(* IEC 61131-3 sources: PortalRobot/Portal_robot/Device/application (part 5) *)

(* ---- PLC_PRG.RunTestControl.st ---- *)
METHOD PRIVATE RunTestControl

// --- BEGIN IMPLEMENTATION ---

// Test environment is independent from the robot control interface.
rtTestEnvironmentApply(CLK := GVL_HMI.xTestEnvironmentApply);
rtTestSpeedProfileApply(CLK := GVL_HMI.xTestSpeedProfileApply);
rtTestScenarioApply(CLK := GVL_HMI.xTestScenarioApply);
xTestInitializePulse := FALSE;
xTestAbortActive := GVL_HMI.xTestAbort
	AND GVL_HMI.xTestSessionActive
	AND (GVL_CELL_SETTINGS.eTestEnvironment = E_CELL_TEST_ENVIRONMENT.SIMULATION);

xTestStable := NOT GVL_CELL_MANAGER.Status.xRunning
	AND NOT GVL_ROBOT.Status.xBusy
	AND NOT GVL_MAGAZINE.astStatus[1].xBusy
	AND NOT GVL_MAGAZINE.astStatus[2].xBusy
	AND NOT GVL_TWO_PALLET.astInput[1].xPowered
	AND NOT GVL_TWO_PALLET.astInput[2].xPowered
	AND NOT xMotionBusy
	AND NOT SIMULATION_DYNAMICS.xBusy;
FOR uiTestIndex := UINT#1 TO UINT#3 DO
	xTestStable := xTestStable
		AND NOT GVL_MACHINE.Status[uiTestIndex].xBusy
		AND NOT GVL_MACHINE.Status[uiTestIndex].xProcessing;
END_FOR;

GVL_HMI.xTestEnvironmentChangeAllowed := xTestStable;
GVL_HMI.xTestScenarioApplyAllowed := xTestStable
	AND (GVL_TWO_PALLET.uiMode = 0) // Existing scenarios describe static 120-slot magazines
	AND GVL_HMI.xTestSessionActive
	AND (GVL_CELL_SETTINGS.eTestEnvironment <> E_CELL_TEST_ENVIRONMENT.NORMAL)
	AND ((GVL_CELL_SETTINGS.eTestEnvironment <> E_CELL_TEST_ENVIRONMENT.SC500_BENCH)
		OR GVL_TEST_IO.xSc500BenchKeyInput)
	AND ((GVL_CELL_SETTINGS.eTestEnvironment <> E_CELL_TEST_ENVIRONMENT.SIMULATION)
		OR NOT GVL_ROBOT_MODBUS.xModeActive
		OR GVL_ROBOT_MODBUS.Status.xSimulatorActive);
GVL_HMI.xSc500BenchKeyActive := GVL_TEST_IO.xSc500BenchKeyInput;

IF rtTestEnvironmentApply.Q THEN
	GVL_HMI.uiTestRejectReason := UINT#0;
	IF NOT GVL_HMI.xTestEnvironmentChangeAllowed THEN
		GVL_HMI.uiTestRejectReason := UINT#1; // equipment is not idle
	ELSIF GVL_HMI.uiTestEnvironmentRequest > UINT#2 THEN
		GVL_HMI.uiTestRejectReason := UINT#2; // invalid environment
	ELSIF (GVL_HMI.uiTestEnvironmentRequest = UINT#2)
	AND (NOT GVL_ROBOT_MODBUS.xModeActive OR NOT GVL_TEST_IO.xSc500BenchKeyInput) THEN
		GVL_HMI.uiTestRejectReason := UINT#3; // bench requires Modbus and physical key
	ELSIF (GVL_HMI.uiTestEnvironmentRequest = UINT#1)
	AND GVL_ROBOT_MODBUS.xModeActive
	AND NOT GVL_ROBOT_MODBUS.Status.xSimulatorActive THEN
		GVL_HMI.uiTestRejectReason := UINT#4; // Python simulator marker missing
	ELSE
		CASE GVL_HMI.uiTestEnvironmentRequest OF
			UINT#0: GVL_CELL_SETTINGS.eTestEnvironment := E_CELL_TEST_ENVIRONMENT.NORMAL;
			UINT#1: GVL_CELL_SETTINGS.eTestEnvironment := E_CELL_TEST_ENVIRONMENT.SIMULATION;
			UINT#2: GVL_CELL_SETTINGS.eTestEnvironment := E_CELL_TEST_ENVIRONMENT.SC500_BENCH;
		END_CASE;
		GVL_CELL_SETTINGS.eTestSpeedProfile := E_TEST_SPEED_PROFILE.REALTIME;
		xSc500BenchKeyLost := FALSE;
	END_IF;
END_IF;

IF rtTestSpeedProfileApply.Q THEN
	GVL_HMI.uiTestRejectReason := UINT#0;
	IF (GVL_HMI.uiTestSpeedProfileRequest <= UINT#1)
	AND (GVL_CELL_SETTINGS.eTestEnvironment = E_CELL_TEST_ENVIRONMENT.SIMULATION) THEN
		IF GVL_HMI.uiTestSpeedProfileRequest = UINT#1 THEN
			GVL_CELL_SETTINGS.eTestSpeedProfile := E_TEST_SPEED_PROFILE.FAST;
			// В Modbus профиль по-прежнему владеет коэффициентом внешней модели.
			// В SoftMotion коэффициент задаёт ползунок, а применение выполняется
			// отдельной транзакцией только на границе следующего теста.
			IF GVL_ROBOT_MODBUS.xModeActive THEN
				GVL_CELL_SETTINGS.uiSimulationTimeFactor := UINT#250;
			END_IF;
		ELSE
			GVL_CELL_SETTINGS.eTestSpeedProfile := E_TEST_SPEED_PROFILE.REALTIME;
			IF GVL_ROBOT_MODBUS.xModeActive THEN
				GVL_CELL_SETTINGS.uiSimulationTimeFactor := UINT#1;
			END_IF;
		END_IF;
		GVL_HMI.uiSimulationTimeFactor := GVL_CELL_SETTINGS.uiSimulationTimeFactor;
	ELSE
		GVL_HMI.uiTestRejectReason := UINT#5; // speed profile is simulation-only
	END_IF;
END_IF;

// Losing the physical key does not interrupt the current SC-500 command.
// As soon as it finishes, robot readiness is removed and no next command can start.
IF (GVL_CELL_SETTINGS.eTestEnvironment = E_CELL_TEST_ENVIRONMENT.SC500_BENCH)
AND NOT GVL_TEST_IO.xSc500BenchKeyInput THEN
	xSc500BenchKeyLost := TRUE;
	IF NOT GVL_ROBOT_MODBUS.Status.xBusy THEN
		xRobotInterfaceReady := FALSE;
		xDrivesReady := FALSE;
	END_IF;
END_IF;

IF rtTestScenarioApply.Q THEN
	GVL_HMI.uiTestScenarioResult := UINT#0;
	xTestScenarioValid := GVL_HMI.stTestScenario.udiLoadSeq <> UDINT#0
		AND (GVL_HMI.stTestScenario.uiTypeCount >= UINT#1)
		AND (GVL_HMI.stTestScenario.uiTypeCount <= UINT#3);
	FOR uiTestIndex := UINT#1 TO UINT#3 DO
		xTestScenarioValid := xTestScenarioValid
			AND (GVL_HMI.stTestScenario.auiMachineState[uiTestIndex] <= UINT#3)
			AND (GVL_HMI.stTestScenario.auiMachineType[uiTestIndex] >= UINT#1)
			AND (GVL_HMI.stTestScenario.auiMachineType[uiTestIndex]
				<= GVL_HMI.stTestScenario.uiTypeCount);
	END_FOR;
	FOR uiTestIndex := UINT#1 TO UINT#120 DO
		xTestScenarioValid := xTestScenarioValid
			AND (GVL_HMI.stTestScenario.auiSlotType[uiTestIndex] >= UINT#1)
			AND (GVL_HMI.stTestScenario.auiSlotType[uiTestIndex]
				<= GVL_HMI.stTestScenario.uiTypeCount);
		FOR uiTestMagazine := UINT#1 TO UINT#2 DO
			xTestScenarioValid := xTestScenarioValid
				AND (GVL_HMI.stTestScenario.aauiSlotContent[uiTestMagazine, uiTestIndex] <= UINT#2);
		END_FOR;
	END_FOR;
	uiTestFaultOwnerCount := UINT#0;
	IF GVL_HMI.stTestScenario.dwCellFaultMask <> DWORD#0 THEN
		uiTestFaultOwnerCount := uiTestFaultOwnerCount + UINT#1;
	END_IF;
	IF GVL_HMI.stTestScenario.dwRobotFaultMask <> DWORD#0 THEN
		uiTestFaultOwnerCount := uiTestFaultOwnerCount + UINT#1;
	END_IF;
	FOR uiTestMagazine := UINT#1 TO UINT#2 DO
		IF GVL_HMI.stTestScenario.adwMagazineFaultMask[uiTestMagazine] <> DWORD#0 THEN
			uiTestFaultOwnerCount := uiTestFaultOwnerCount + UINT#1;
		END_IF;
		xTestScenarioValid := xTestScenarioValid
			AND (GVL_HMI.stTestScenario.adwMagazineFaultMask[uiTestMagazine] <= DWORD#16#0000_003F);
	END_FOR;
	FOR uiTestIndex := UINT#1 TO UINT#3 DO
		IF GVL_HMI.stTestScenario.adwMachineFaultMask[uiTestIndex] <> DWORD#0 THEN
			uiTestFaultOwnerCount := uiTestFaultOwnerCount + UINT#1;
		END_IF;
		xTestScenarioValid := xTestScenarioValid
			AND (GVL_HMI.stTestScenario.adwMachineFaultMask[uiTestIndex] <= DWORD#16#0000_07FF);
	END_FOR;
	xTestScenarioValid := xTestScenarioValid
		AND (uiTestFaultOwnerCount <= UINT#1)
		AND (GVL_HMI.stTestScenario.dwCellFaultMask <= DWORD#16#0000_0001)
		AND (GVL_HMI.stTestScenario.dwRobotFaultMask <= DWORD#16#0000_01FF)
		AND (GVL_HMI.stTestScenario.auiGripperContent[1] <= UINT#1)
		AND ((GVL_HMI.stTestScenario.auiGripperContent[1] = UINT#0)
			= (GVL_HMI.stTestScenario.auiGripperType[1] = UINT#0))
		AND (GVL_HMI.stTestScenario.auiGripperType[1]
			<= GVL_HMI.stTestScenario.uiTypeCount)
		AND ((GVL_HMI.stTestScenario.auiGripperContent[2] = UINT#0)
			OR (GVL_HMI.stTestScenario.auiGripperContent[2] = UINT#2))
		AND ((GVL_HMI.stTestScenario.auiGripperContent[2] = UINT#0)
			= (GVL_HMI.stTestScenario.auiGripperType[2] = UINT#0))
		AND (GVL_HMI.stTestScenario.auiGripperType[2]
			<= GVL_HMI.stTestScenario.uiTypeCount);

	IF NOT GVL_HMI.xTestScenarioApplyAllowed THEN
		GVL_HMI.uiTestScenarioResult := UINT#1;
	ELSIF NOT xTestScenarioValid OR (GVL_HMI.stTestScenario.uiOrientation > UINT#1) THEN
		GVL_HMI.uiTestScenarioResult := UINT#2;
	ELSE
		FOR uiTestMagazine := UINT#1 TO UINT#2 DO
			FOR uiTestIndex := UINT#1 TO UINT#120 DO
				GVL_DETAIL.astMagazine[uiTestMagazine].aSlots[uiTestIndex].xInPosition :=
					GVL_HMI.stTestScenario.aauiSlotContent[uiTestMagazine, uiTestIndex] <> UINT#0;
				CASE GVL_HMI.stTestScenario.aauiSlotContent[uiTestMagazine, uiTestIndex] OF
					UINT#1: GVL_DETAIL.astMagazine[uiTestMagazine].aSlots[uiTestIndex].eDetailType := E_DETAIL_TYPE.BLANK;
					UINT#2: GVL_DETAIL.astMagazine[uiTestMagazine].aSlots[uiTestIndex].eDetailType := E_DETAIL_TYPE.DETAIL;
				ELSE
					GVL_DETAIL.astMagazine[uiTestMagazine].aSlots[uiTestIndex].eDetailType := E_DETAIL_TYPE.NONE;
				END_CASE;
				IF GVL_HMI.stTestScenario.aauiSlotContent[uiTestMagazine, uiTestIndex] = UINT#0 THEN
					GVL_DETAIL.astMagazine[uiTestMagazine].aSlots[uiTestIndex].uiProductType := UINT#0;
				ELSE
					GVL_DETAIL.astMagazine[uiTestMagazine].aSlots[uiTestIndex].uiProductType :=
						GVL_HMI.stTestScenario.auiSlotType[uiTestIndex];
				END_IF;
			END_FOR;
			adwTestMagazineFaultMask[uiTestMagazine] :=
				GVL_HMI.stTestScenario.adwMagazineFaultMask[uiTestMagazine];
		END_FOR;
		// Начальные инъекции: маски переводятся в существующий диагностический
		// контракт, а не обходят владельцев ошибок.
		axHmiInternalPulse[13] :=
			(GVL_HMI.stTestScenario.dwCellFaultMask AND DWORD#16#0000_0001) <> DWORD#0;
		axHmiInternalPulse[12] :=
			(GVL_HMI.stTestScenario.dwRobotFaultMask AND DWORD#16#0000_0001) <> DWORD#0;
		GVL_HMI.xSimGripper1Fault :=
			(GVL_HMI.stTestScenario.dwRobotFaultMask AND DWORD#16#0000_0002) <> DWORD#0;
		GVL_HMI.xSimGripper2Fault :=
			(GVL_HMI.stTestScenario.dwRobotFaultMask AND DWORD#16#0000_0004) <> DWORD#0;
		GVL_HMI.xSimGripperRotationFault :=
			(GVL_HMI.stTestScenario.dwRobotFaultMask AND DWORD#16#0000_0008) <> DWORD#0;
		GVL_HMI.xSimGripperGlobalFault :=
			(GVL_HMI.stTestScenario.dwRobotFaultMask AND DWORD#16#0000_0010) <> DWORD#0;
		axHmiInternalPulse[14] :=
			(GVL_HMI.stTestScenario.dwRobotFaultMask AND DWORD#16#0000_0020) <> DWORD#0;
		axHmiInternalPulse[15] :=
			(GVL_HMI.stTestScenario.dwRobotFaultMask AND DWORD#16#0000_0040) <> DWORD#0;
		axHmiInternalPulse[16] :=
			(GVL_HMI.stTestScenario.dwRobotFaultMask AND DWORD#16#0000_0080) <> DWORD#0;
		axHmiInternalPulse[17] :=
			(GVL_HMI.stTestScenario.dwRobotFaultMask AND DWORD#16#0000_0100) <> DWORD#0;
		axHmiInternalPulse[18] :=
			(GVL_HMI.stTestScenario.adwMagazineFaultMask[1] AND DWORD#16#0000_0001) <> DWORD#0;
		axHmiInternalPulse[19] :=
			(GVL_HMI.stTestScenario.adwMagazineFaultMask[1] AND DWORD#16#0000_0002) <> DWORD#0;
		axHmiInternalPulse[20] :=
			(GVL_HMI.stTestScenario.adwMagazineFaultMask[1] AND DWORD#16#0000_0004) <> DWORD#0;
		axHmiInternalPulse[21] :=
			(GVL_HMI.stTestScenario.adwMagazineFaultMask[1] AND DWORD#16#0000_0008) <> DWORD#0;
		axHmiInternalPulse[22] :=
			(GVL_HMI.stTestScenario.adwMagazineFaultMask[1] AND DWORD#16#0000_0010) <> DWORD#0;
		axHmiInternalPulse[23] :=
			(GVL_HMI.stTestScenario.adwMagazineFaultMask[1] AND DWORD#16#0000_0020) <> DWORD#0;
		FOR uiTestIndex := UINT#1 TO UINT#3 DO
			GVL_HMI.axMachineSimAlarm[uiTestIndex] :=
				(GVL_HMI.stTestScenario.adwMachineFaultMask[uiTestIndex] AND DWORD#16#0000_0001) <> DWORD#0;
			GVL_HMI.axMachineSimDoorFault[uiTestIndex] :=
				(GVL_HMI.stTestScenario.adwMachineFaultMask[uiTestIndex] AND DWORD#16#0000_0002) <> DWORD#0;
			GVL_HMI.axMachineSimChuckFault[uiTestIndex] :=
				(GVL_HMI.stTestScenario.adwMachineFaultMask[uiTestIndex] AND DWORD#16#0000_0004) <> DWORD#0;
			GVL_HMI.axMachineTimeoutRobotMove[uiTestIndex] :=
				(GVL_HMI.stTestScenario.adwMachineFaultMask[uiTestIndex] AND DWORD#16#0000_0008) <> DWORD#0;
			GVL_HMI.axMachineTimeoutRobotAction[uiTestIndex] :=
				(GVL_HMI.stTestScenario.adwMachineFaultMask[uiTestIndex] AND DWORD#16#0000_0010) <> DWORD#0;
			GVL_HMI.axMachineTimeoutRobotRelease[uiTestIndex] :=
				(GVL_HMI.stTestScenario.adwMachineFaultMask[uiTestIndex] AND DWORD#16#0000_0020) <> DWORD#0;
			GVL_HMI.axMachineTimeoutDoorOpen[uiTestIndex] :=
				(GVL_HMI.stTestScenario.adwMachineFaultMask[uiTestIndex] AND DWORD#16#0000_0040) <> DWORD#0;
			GVL_HMI.axMachineTimeoutDoorClose[uiTestIndex] :=
				(GVL_HMI.stTestScenario.adwMachineFaultMask[uiTestIndex] AND DWORD#16#0000_0080) <> DWORD#0;
			GVL_HMI.axMachineTimeoutChuckOpen[uiTestIndex] :=
				(GVL_HMI.stTestScenario.adwMachineFaultMask[uiTestIndex] AND DWORD#16#0000_0100) <> DWORD#0;
			GVL_HMI.axMachineTimeoutChuckClose[uiTestIndex] :=
				(GVL_HMI.stTestScenario.adwMachineFaultMask[uiTestIndex] AND DWORD#16#0000_0200) <> DWORD#0;
			GVL_HMI.axMachineTimeoutCycleStart[uiTestIndex] :=
				(GVL_HMI.stTestScenario.adwMachineFaultMask[uiTestIndex] AND DWORD#16#0000_0400) <> DWORD#0;
		END_FOR;
		GVL_HMI.xErrorSimulationEnable :=
			(GVL_HMI.stTestScenario.dwCellFaultMask <> DWORD#0)
			OR (GVL_HMI.stTestScenario.dwRobotFaultMask <> DWORD#0)
			OR (GVL_HMI.stTestScenario.adwMagazineFaultMask[1] <> DWORD#0)
			OR (GVL_HMI.stTestScenario.adwMagazineFaultMask[2] <> DWORD#0)
			OR (GVL_HMI.stTestScenario.adwMachineFaultMask[1] <> DWORD#0)
			OR (GVL_HMI.stTestScenario.adwMachineFaultMask[2] <> DWORD#0)
			OR (GVL_HMI.stTestScenario.adwMachineFaultMask[3] <> DWORD#0);
		xTestInitializePulse := TRUE;
	END_IF;
	// Ack подтверждает обработку конкретного LoadSeq даже при отклонении.
	GVL_HMI.udiTestScenarioAckSeq := GVL_HMI.stTestScenario.udiLoadSeq;
END_IF;

GVL_HMI.uiTestEnvironmentApplied := TO_UINT(GVL_CELL_SETTINGS.eTestEnvironment);
GVL_HMI.uiTestSpeedProfileApplied := TO_UINT(GVL_CELL_SETTINGS.eTestSpeedProfile);
GVL_HMI.xSc500BenchKeyLost := xSc500BenchKeyLost;
IF GVL_CELL_SETTINGS.eTestEnvironment = E_CELL_TEST_ENVIRONMENT.SIMULATION THEN
	IF GVL_HMI.xTestSessionActive THEN
		GVL_CELL_SETTINGS.xSimulationAccelerationEnable :=
			GVL_CELL_SETTINGS.eTestSpeedProfile = E_TEST_SPEED_PROFILE.FAST;
		// Профиль владеет включением ускоренных таймеров, а сам коэффициент
		// разрешено менять с HMI прямо во время тестового движения.
		GVL_HMI.xSimulationAccelerationEnable := GVL_CELL_SETTINGS.xSimulationAccelerationEnable;
	END_IF;
ELSE
	GVL_CELL_SETTINGS.xSimulationAccelerationEnable := FALSE;
	GVL_HMI.xSimulationAccelerationEnable := FALSE;
END_IF;

(* ---- PLC_PRG.RunTwoPallet.st ---- *)
METHOD PRIVATE RunTwoPallet

// --- BEGIN IMPLEMENTATION ---

GVL_TWO_PALLET.xModeChanged := FALSE;
IF NOT xTwinSimulationInitialized THEN
	FOR uiTwin := 1 TO 2 DO
		// Числа используются только для виртуальных SoftMotion-осей.
		GVL_TWO_PALLET.astSimulationConfig[uiTwin].xConfigured := TRUE;
		GVL_TWO_PALLET.astSimulationConfig[uiTwin].xP1LockOut := TRUE;
		GVL_TWO_PALLET.axSimulationAutoSwapEnabled[uiTwin] := TRUE;
		GVL_TWO_PALLET.astSimulationConfig[uiTwin].lrExchange := 0.0;
		GVL_TWO_PALLET.astSimulationConfig[uiTwin].lrWorkP1 := 100.0;
		GVL_TWO_PALLET.astSimulationConfig[uiTwin].lrWorkP2 := 200.0;
		GVL_TWO_PALLET.astSimulationConfig[uiTwin].lrHome := 0.0;
		GVL_TWO_PALLET.astSimulationConfig[uiTwin].lrTolerance := 1.0;
		GVL_TWO_PALLET.astSimulationConfig[uiTwin].lrVelocity := 100.0;
		GVL_TWO_PALLET.astSimulationConfig[uiTwin].lrAcceleration := 200.0;
		GVL_TWO_PALLET.astSimulationConfig[uiTwin].lrDeceleration := 200.0;
		GVL_TWO_PALLET.astSimulationConfig[uiTwin].lrJerk := 1000.0;
		GVL_TWO_PALLET.astSimulationConfig[uiTwin].tCylinder := T#3S;
		GVL_TWO_PALLET.astSimulationConfig[uiTwin].tMove := T#20S;
		GVL_TWO_PALLET.astSimulationConfig[uiTwin].tHome := T#10S;
		GVL_TWO_PALLET.astSimulationConfig[uiTwin].tPulse := T#150MS;
	END_FOR;
	IF NOT GVL_TWO_PALLET.xAutoSwapDefaultsApplied THEN
		FOR uiTwin := 1 TO 2 DO
			GVL_TWO_PALLET.axAutoSwapEnabled[uiTwin] := TRUE;
		END_FOR;
		GVL_TWO_PALLET.xAutoSwapDefaultsApplied := TRUE;
	END_IF;
	xTwinSimulationInitialized := TRUE;
END_IF;
FOR uiTwin := 1 TO 2 DO
	GVL_TWO_PALLET.auiCommand[uiTwin] := UINT#0;
END_FOR;
IF NOT xTwinStartup THEN
	IF GVL_TWO_PALLET.uiMode = 0 THEN
		GVL_HMI.MagazinePitchX := GVL_TWO_PALLET.lrStaticPitchX;
		GVL_HMI.MagazinePitchY := GVL_TWO_PALLET.lrStaticPitchY;
	ELSE
		GVL_HMI.MagazinePitchX := GVL_TWO_PALLET.lrTwinPitchX;
		GVL_HMI.MagazinePitchY := GVL_TWO_PALLET.lrTwinPitchY;
	END_IF;
	FOR uiTwin := 1 TO 2 DO
		// После перезапуска содержимое сохранено, готовность загрузки подтверждается заново.
		GVL_TWO_PALLET.astStore[uiTwin].axLoaded[1] := FALSE;
		GVL_TWO_PALLET.astStore[uiTwin].axLoaded[2] := FALSE;
		IF GVL_TWO_PALLET.uiMode = 0 THEN
			GVL_DETAIL.astMagazine[uiTwin] := GVL_TWO_PALLET.astStatic[uiTwin];
		END_IF;
	END_FOR;
	xTwinStartup := TRUE;
END_IF;
GVL_TWO_PALLET.xModeChangeAllowed := GVL_CELL_CONTROL.xManual
	AND NOT GVL_CELL_MANAGER.Status.xRunning AND NOT GVL_ROBOT.Status.xBusy AND NOT xMotionBusy
	AND xHmiConnectionAlive AND NOT GVL_HMI.xTestSessionActive AND NOT GVL_ROBOT.Status.xBlankAvailable AND NOT GVL_ROBOT.Status.xDetailAvailable
	AND (GVL_ROBOT.Status.uiMagazineContext = 0)
	AND NOT GVL_MAGAZINE.astStatus[1].xEnabled AND NOT GVL_MAGAZINE.astStatus[2].xEnabled
	AND NOT GVL_MAGAZINE.astStatus[1].xBusy AND NOT GVL_MAGAZINE.astStatus[2].xBusy
	AND NOT GVL_TWO_PALLET.astStatus[1].xBusy AND NOT GVL_TWO_PALLET.astStatus[2].xBusy
	AND NOT GVL_TWO_PALLET.astInput[1].xPowered AND NOT GVL_TWO_PALLET.astInput[2].xPowered
	AND NOT GVL_TWO_PALLET.astStatus[1].xError AND NOT GVL_TWO_PALLET.astStatus[2].xError;

udiTwinSnapshot := GVL_HMI.udiTwinCommandSeq;
uiTwinRequestResult := 0;
xTwinInventoryCommand := FALSE;
IF (udiTwinSnapshot <> 0) AND (udiTwinSnapshot <> GVL_HMI.udiTwinAckSeq) THEN
	stTwinRequest := GVL_HMI.stTwinRequest;
	uiTwinRequestResult := 2; // Условие команды не выполнено
	IF (GVL_HMI.udiHmiCommandClockMs - GVL_HMI.udiTwinIssuedAtMs) > 2000 THEN
		uiTwinRequestResult := 4;
	ELSIF (stTwinRequest.uiMagazine = 0) AND (stTwinRequest.uiCommand = 25) THEN
		IF GVL_TWO_PALLET.xModeChangeAllowed AND (stTwinRequest.uiValue <= 1) AND xHmiConnectionAlive THEN
			IF GVL_TWO_PALLET.uiMode <> stTwinRequest.uiValue THEN
				IF GVL_TWO_PALLET.uiMode = 0 THEN
					GVL_TWO_PALLET.lrStaticPitchX := GVL_HMI.MagazinePitchX;
					GVL_TWO_PALLET.lrStaticPitchY := GVL_HMI.MagazinePitchY;
				ELSE
					GVL_TWO_PALLET.lrTwinPitchX := GVL_HMI.MagazinePitchX;
					GVL_TWO_PALLET.lrTwinPitchY := GVL_HMI.MagazinePitchY;
				END_IF;
				GVL_TWO_PALLET.uiMode := stTwinRequest.uiValue;
				GVL_TWO_PALLET.xModeChanged := TRUE;
				FOR uiTwin := 1 TO 2 DO
					IF GVL_TWO_PALLET.uiMode = 0 THEN GVL_DETAIL.astMagazine[uiTwin] := GVL_TWO_PALLET.astStatic[uiTwin]; END_IF;
					// Базы меняются вместе с механикой: старые координаты нельзя молча использовать.
					GVL_POINT.astRetainPoints[13 + uiTwin].xConfigured := FALSE;
				END_FOR;
				IF GVL_TWO_PALLET.uiMode = 0 THEN
					GVL_HMI.MagazinePitchX := GVL_TWO_PALLET.lrStaticPitchX; GVL_HMI.MagazinePitchY := GVL_TWO_PALLET.lrStaticPitchY;
				ELSE
					GVL_HMI.MagazinePitchX := GVL_TWO_PALLET.lrTwinPitchX; GVL_HMI.MagazinePitchY := GVL_TWO_PALLET.lrTwinPitchY;
				END_IF;
				xPointTableReady := FALSE;
			END_IF;
			uiTwinRequestResult := 1;
		END_IF;
	ELSIF (stTwinRequest.uiMagazine >= 1) AND (stTwinRequest.uiMagazine <= 2)
		AND (GVL_TWO_PALLET.uiMode = 1) THEN
		uiTwin := stTwinRequest.uiMagazine;
		IF ((stTwinRequest.uiCommand >= 1) AND (stTwinRequest.uiCommand <= 19))
			OR ((stTwinRequest.uiCommand >= 25) AND (stTwinRequest.uiCommand <= 32)) THEN
			GVL_TWO_PALLET.auiCommand[uiTwin] := stTwinRequest.uiCommand;
			GVL_TWO_PALLET.auiValue[uiTwin] := stTwinRequest.uiValue;
			GVL_TWO_PALLET.audiRevision[uiTwin] := stTwinRequest.udiRevision;
		ELSIF (stTwinRequest.uiCommand >= UINT#20)
			AND (stTwinRequest.uiCommand <= UINT#24) THEN
			xTwinInventoryCommand := TRUE; // Проверить по разрешениям текущего скана ПОСЛЕ вызова FB
		ELSIF stTwinRequest.uiCommand = UINT#33 THEN
			IF (stTwinRequest.uiValue <= UINT#1) AND xHmiConnectionAlive THEN
				IF GVL_CELL_SETTINGS.eTestEnvironment = E_CELL_TEST_ENVIRONMENT.SIMULATION THEN
					GVL_TWO_PALLET.axSimulationAutoSwapEnabled[uiTwin] := stTwinRequest.uiValue = UINT#1;
				ELSE
					GVL_TWO_PALLET.axAutoSwapEnabled[uiTwin] := stTwinRequest.uiValue = UINT#1;
				END_IF;
				uiTwinRequestResult := UINT#1;
			END_IF;
		END_IF;
	END_IF;
END_IF;

FOR uiTwin := 1 TO 2 DO
	GVL_TWO_PALLET.astActiveConfig[uiTwin] := GVL_TWO_PALLET.astConfig[uiTwin];
	IF GVL_CELL_SETTINGS.eTestEnvironment = E_CELL_TEST_ENVIRONMENT.SIMULATION THEN
		GVL_TWO_PALLET.astActiveConfig[uiTwin] := GVL_TWO_PALLET.astSimulationConfig[uiTwin];
		xTwinAutoSwapEnabled := GVL_TWO_PALLET.axSimulationAutoSwapEnabled[uiTwin];
	ELSE
		xTwinAutoSwapEnabled := GVL_TWO_PALLET.axAutoSwapEnabled[uiTwin];
	END_IF;
	// Старые RETAIN-параметры сохраняют прежнюю полярность до первой настройки
	// полных сочетаний. Нормализуем только рабочую копию, без записи в RETAIN.
	IF NOT GVL_TWO_PALLET.astActiveConfig[uiTwin].xSignalPatternsConfigured THEN
		GVL_TWO_PALLET.astActiveConfig[uiTwin].uiP1Signals := UINT#38;
		GVL_TWO_PALLET.astActiveConfig[uiTwin].uiP2Signals := UINT#26;
		IF GVL_TWO_PALLET.astActiveConfig[uiTwin].xP1LockOut THEN
			GVL_TWO_PALLET.astActiveConfig[uiTwin].uiP1Signals := UINT#26;
			GVL_TWO_PALLET.astActiveConfig[uiTwin].uiP2Signals := UINT#38;
		END_IF;
		GVL_TWO_PALLET.astActiveConfig[uiTwin].xSignalPatternsConfigured := TRUE;
	END_IF;
	// Legacy power/reset также проходит владельца механизма и его блокировки.
	IF (GVL_TWO_PALLET.auiCommand[uiTwin] = 0) AND (GVL_TWO_PALLET.uiMode = 1) THEN
		IF GVL_HMI.astMagazineCommand[uiTwin].xEnable THEN GVL_TWO_PALLET.auiCommand[uiTwin] := 1; END_IF;
		IF GVL_HMI.astMagazineCommand[uiTwin].xDisable OR GVL_CELL_CONTROL.xDisable THEN GVL_TWO_PALLET.auiCommand[uiTwin] := 3; END_IF;
		IF GVL_HMI.astMagazineCommand[uiTwin].xStop THEN GVL_TWO_PALLET.auiCommand[uiTwin] := 15; END_IF;
		IF GVL_HMI.astMagazineCommand[uiTwin].xReset
			OR (GVL_CELL_CONTROL.xReset AND GVL_TWO_PALLET.astStatus[uiTwin].xResetAllowed) THEN
			GVL_TWO_PALLET.auiCommand[uiTwin] := 16;
		END_IF;
	END_IF;

	// Единственное место преобразования транспортных номеров HMI в интерфейс FB.
	astTwinCommand[uiTwin].xEnable := GVL_TWO_PALLET.auiCommand[uiTwin] = UINT#1;
	astTwinCommand[uiTwin].xConfirm := GVL_TWO_PALLET.auiCommand[uiTwin] = UINT#2;
	astTwinCommand[uiTwin].xStart := GVL_TWO_PALLET.auiCommand[uiTwin] = UINT#27;
	astTwinCommand[uiTwin].xRejectStart := GVL_TWO_PALLET.auiCommand[uiTwin] = UINT#28;
	astTwinCommand[uiTwin].xDisable := GVL_TWO_PALLET.auiCommand[uiTwin] = UINT#3;
	astTwinCommand[uiTwin].xSwap := GVL_TWO_PALLET.auiCommand[uiTwin] = UINT#4;
	astTwinCommand[uiTwin].xPowerOn := GVL_TWO_PALLET.auiCommand[uiTwin] = UINT#5;
	astTwinCommand[uiTwin].xPowerOff := GVL_TWO_PALLET.auiCommand[uiTwin] = UINT#6;
	astTwinCommand[uiTwin].xDriveReset := GVL_TWO_PALLET.auiCommand[uiTwin] = UINT#7;
	astTwinCommand[uiTwin].xHome := GVL_TWO_PALLET.auiCommand[uiTwin] = UINT#8;
	astTwinCommand[uiTwin].xLower := GVL_TWO_PALLET.auiCommand[uiTwin] = UINT#9;
	astTwinCommand[uiTwin].xRaise := GVL_TWO_PALLET.auiCommand[uiTwin] = UINT#10;
	astTwinCommand[uiTwin].xSelectPallet := (GVL_TWO_PALLET.auiCommand[uiTwin] = UINT#11)
		OR (GVL_TWO_PALLET.auiCommand[uiTwin] = UINT#12);
	astTwinCommand[uiTwin].xLockIn := GVL_TWO_PALLET.auiCommand[uiTwin] = UINT#29;
	astTwinCommand[uiTwin].xLockOut := GVL_TWO_PALLET.auiCommand[uiTwin] = UINT#30;
	astTwinCommand[uiTwin].xStopIn := GVL_TWO_PALLET.auiCommand[uiTwin] = UINT#31;
	astTwinCommand[uiTwin].xStopOut := GVL_TWO_PALLET.auiCommand[uiTwin] = UINT#32;
	astTwinCommand[uiTwin].xMoveToExchange := GVL_TWO_PALLET.auiCommand[uiTwin] = UINT#13;
	astTwinCommand[uiTwin].xMoveToWork := GVL_TWO_PALLET.auiCommand[uiTwin] = UINT#14;
	astTwinCommand[uiTwin].xStop := GVL_TWO_PALLET.auiCommand[uiTwin] = UINT#15;
	astTwinCommand[uiTwin].xReset := GVL_TWO_PALLET.auiCommand[uiTwin] = UINT#16;
	astTwinCommand[uiTwin].xJogPositive := GVL_TWO_PALLET.auiCommand[uiTwin] = UINT#17;
	astTwinCommand[uiTwin].xJogNegative := GVL_TWO_PALLET.auiCommand[uiTwin] = UINT#18;
	astTwinCommand[uiTwin].xJogRelease := GVL_TWO_PALLET.auiCommand[uiTwin] = UINT#19;
	astTwinCommand[uiTwin].xTeachOperator := GVL_TWO_PALLET.auiCommand[uiTwin] = UINT#25;
	astTwinCommand[uiTwin].xTeachWork := GVL_TWO_PALLET.auiCommand[uiTwin] = UINT#26;
	astTwinCommand[uiTwin].uiPallet := GVL_TWO_PALLET.auiValue[uiTwin];
	IF GVL_TWO_PALLET.auiCommand[uiTwin] = UINT#11 THEN
		astTwinCommand[uiTwin].uiPallet := UINT#1;
	ELSIF GVL_TWO_PALLET.auiCommand[uiTwin] = UINT#12 THEN
		astTwinCommand[uiTwin].uiPallet := UINT#2;
	END_IF;
	astTwinCommand[uiTwin].udiRevision := GVL_TWO_PALLET.audiRevision[uiTwin];

	// xBusy не покрывает удерживаемый запрос и завершение Disable.
	// Занятость другого магазина/станка сама по себе не запрещает правку инвентаря.
	xTwinRobotOperation := GVL_MAGAZINE.astPartStatus[uiTwin].xBusy
		OR GVL_MAGAZINE.astPartStatus[uiTwin].xDisablePending
		OR GVL_MAGAZINE.astAutoCommand[uiTwin].xExecute
		OR GVL_MAGAZINE.astCommand[uiTwin].xExecute
		OR ((GVL_ROBOT.Status.xBusy OR xMotionBusy)
			AND (GVL_ROBOT.Status.uiMagazineContext = uiTwin));
	xTwinRobotClear := NOT GVL_ROBOT.Status.xBusy AND NOT xMotionBusy
		AND NOT xTwinRobotOperation
		AND GVL_CELL_MANAGER.Status.xMagazineExchangeAllowed
		AND NOT GVL_MACHINE.Status[1].xBusy AND NOT GVL_MACHINE.Status[2].xBusy AND NOT GVL_MACHINE.Status[3].xBusy
		AND NOT GVL_ROBOT.Status.xError AND xRobotInterfaceReady
		AND (GVL_ROBOT.Status.eCurrentPoint <> E_POINT_NAME.NONE)
		AND (GVL_ROBOT.Status.uiMagazineContext <> uiTwin)
		AND (GVL_ROBOT.Status.eCurrentPoint <> E_POINT_NAME.MAGAZINE_CHANGE)
		AND (GVL_ROBOT.Status.eCurrentPoint <> E_POINT_NAME.MAGAZINE_IN_SLOT);
	xTwinOtherLoaded := FALSE;
	IF (GVL_TWO_PALLET.astStatus[uiTwin].uiRobotPallet >= UINT#1)
		AND (GVL_TWO_PALLET.astStatus[uiTwin].uiRobotPallet <= UINT#2) THEN
		uiTwinPallet := UINT#3 - GVL_TWO_PALLET.astStatus[uiTwin].uiRobotPallet;
		xTwinOtherLoaded := GVL_TWO_PALLET.astStore[uiTwin].axLoaded[uiTwinPallet];
	END_IF;
	// Запрос сохраняет цикл, пока робот и автоматы освобождают окно обмена.
	// Готовность зоны проверяет FB_TWO_PALLET; она не должна терять сам запрос.
	axTwinAutoSwapPending[uiTwin] := (GVL_TWO_PALLET.uiMode = UINT#1)
		AND GVL_CELL_MANAGER.Status.xRunning
		AND NOT GVL_CELL_MANAGER.Status.xStopPending
		AND NOT GVL_CELL_CONTROL.xStop
		AND NOT GVL_CELL_CONTROL.xManual
		AND GVL_MAGAZINE.astPartStatus[uiTwin].xFinished
		AND xTwinAutoSwapEnabled
		AND xTwinOtherLoaded
		AND NOT astTwinCommand[uiTwin].xDisable
		AND NOT astTwinCommand[uiTwin].xStop;
	TWIN[uiTwin](
		xSelected := GVL_TWO_PALLET.uiMode = 1,
		xManual := GVL_CELL_CONTROL.xManual AND NOT GVL_CELL_MANAGER.Status.xRunning,
		xSafe := CELL_SAFETY.Status.xReady AND NOT GVL_CELL_CONTROL.xGlobalError
			AND CELL_SAFETY.astEnclosureDoorStatus[uiTwin * 2 - 1].xLocked
			AND CELL_SAFETY.astEnclosureDoorStatus[uiTwin * 2].xLocked
			AND NOT CELL_SAFETY.astEnclosureDoorStatus[uiTwin * 2 - 1].xUnlockOutput
			AND NOT CELL_SAFETY.astEnclosureDoorStatus[uiTwin * 2].xUnlockOutput,
		xRobotClear := xTwinRobotClear,
		xRobotIdle := NOT GVL_ROBOT.Status.xBusy AND NOT xMotionBusy,
		xRobotOperation := xTwinRobotOperation,
		xRobotGeometryReady := NOT GVL_HMI.xModbusMode AND xPointTableReady,
		xRobotMagazineReady := GVL_MAGAZINE.astPartStatus[uiTwin].xEnableCheckNoError
			AND GVL_MAGAZINE.astPartStatus[uiTwin].xEnableCheckGeometry,
		xConnection := xHmiConnectionAlive,
		xStopRequest := GVL_CELL_CONTROL.xStop OR GVL_HMI.astMagazineCommand[uiTwin].xStop OR GVL_TWO_PALLET.xModeChanged,
		xAutoSwap := axTwinAutoSwapPending[uiTwin],
		xOtherLoaded := xTwinOtherLoaded,
		xActivePalletEditAllowed := NOT xTwinRobotOperation,
		xConfigurationChanged := axTwinConfigurationChanged[uiTwin],
		xExternalCommandRejected := axTwinExternalCommandRejected[uiTwin],
		Command := astTwinCommand[uiTwin],
		Config := GVL_TWO_PALLET.astActiveConfig[uiTwin], Input := GVL_TWO_PALLET.astInput[uiTwin],
		Status => GVL_TWO_PALLET.astStatus[uiTwin],
		Diag => GVL_TWO_PALLET.astDiag[uiTwin],
		Error => GVL_TWO_PALLET.astError[uiTwin],
		Output => GVL_TWO_PALLET.astOutput[uiTwin]);
	GVL_TWO_PALLET.astStatus[uiTwin].xAutoSwapEnabled := xTwinAutoSwapEnabled;
	// После Disable, Stop или аварии ожидание обмена не удерживает планировщик.
	axTwinAutoSwapPending[uiTwin] := axTwinAutoSwapPending[uiTwin]
		AND GVL_TWO_PALLET.astStatus[uiTwin].xEnabled
		AND NOT GVL_TWO_PALLET.astStatus[uiTwin].xError;
	axTwinConfigurationChanged[uiTwin] := FALSE;
	axTwinExternalCommandRejected[uiTwin] := FALSE;
	IF GVL_TWO_PALLET.astOutput[uiTwin].xTeachOperator THEN
		IF GVL_CELL_SETTINGS.eTestEnvironment = E_CELL_TEST_ENVIRONMENT.SIMULATION THEN
			GVL_TWO_PALLET.astSimulationConfig[uiTwin].lrExchange := GVL_TWO_PALLET.astInput[uiTwin].lrPosition;
		ELSE
			GVL_TWO_PALLET.astConfig[uiTwin].lrExchange := GVL_TWO_PALLET.astInput[uiTwin].lrPosition;
		END_IF;
		axTwinConfigurationChanged[uiTwin] := TRUE;
	END_IF;
	IF GVL_TWO_PALLET.astOutput[uiTwin].xTeachWork THEN
		IF GVL_TWO_PALLET.astStatus[uiTwin].uiSelected = UINT#1 THEN
			IF GVL_CELL_SETTINGS.eTestEnvironment = E_CELL_TEST_ENVIRONMENT.SIMULATION THEN
				GVL_TWO_PALLET.astSimulationConfig[uiTwin].lrWorkP1 := GVL_TWO_PALLET.astInput[uiTwin].lrPosition;
			ELSE
				GVL_TWO_PALLET.astConfig[uiTwin].lrWorkP1 := GVL_TWO_PALLET.astInput[uiTwin].lrPosition;
			END_IF;
		ELSIF GVL_TWO_PALLET.astStatus[uiTwin].uiSelected = UINT#2 THEN
			IF GVL_CELL_SETTINGS.eTestEnvironment = E_CELL_TEST_ENVIRONMENT.SIMULATION THEN
				GVL_TWO_PALLET.astSimulationConfig[uiTwin].lrWorkP2 := GVL_TWO_PALLET.astInput[uiTwin].lrPosition;
			ELSE
				GVL_TWO_PALLET.astConfig[uiTwin].lrWorkP2 := GVL_TWO_PALLET.astInput[uiTwin].lrPosition;
			END_IF;
		END_IF;
		axTwinConfigurationChanged[uiTwin] := TRUE;
	END_IF;
	// RunCellControl ниже должен видеть запрет уже в скане начала обмена.
	IF GVL_TWO_PALLET.uiMode = 1 THEN
		GVL_MAGAZINE.astStatus[uiTwin].xReady := GVL_MAGAZINE.astPartStatus[uiTwin].xReady
			AND GVL_TWO_PALLET.astStatus[uiTwin].xReady;
		GVL_MAGAZINE.astStatus[uiTwin].xBusy := GVL_MAGAZINE.astPartStatus[uiTwin].xBusy
			OR GVL_TWO_PALLET.astStatus[uiTwin].xBusy;
		GVL_MAGAZINE.astStatus[uiTwin].xEnabled := GVL_TWO_PALLET.astStatus[uiTwin].xEnabled;
	END_IF;
	IF GVL_TWO_PALLET.astStatus[uiTwin].xCompleted THEN
		GVL_TWO_PALLET.astStore[uiTwin].axLoaded[1] := FALSE;
		GVL_TWO_PALLET.astStore[uiTwin].axLoaded[2] := FALSE;
	END_IF;
	IF (uiTwinRequestResult = 2) AND (stTwinRequest.uiMagazine = uiTwin)
		AND (((stTwinRequest.uiCommand >= 1) AND (stTwinRequest.uiCommand <= 19))
			OR ((stTwinRequest.uiCommand >= 25) AND (stTwinRequest.uiCommand <= 32)))
		AND GVL_TWO_PALLET.astStatus[uiTwin].xCommandAccepted THEN uiTwinRequestResult := 1; END_IF;
END_FOR;

IF xTwinInventoryCommand THEN
	uiTwin := stTwinRequest.uiMagazine;
	uiTwinPallet := stTwinRequest.uiValue;
	IF stTwinRequest.uiCommand = UINT#24 THEN
		IF GVL_TWO_PALLET.astStatus[uiTwin].xConfigAllowed
			AND stTwinRequest.Config.xSignalPatternsConfigured
			AND TWIN[uiTwin].IsSignalConfigurationValid(
				uiP1Signals := stTwinRequest.Config.uiP1Signals,
				uiP2Signals := stTwinRequest.Config.uiP2Signals) THEN
			IF GVL_CELL_SETTINGS.eTestEnvironment = E_CELL_TEST_ENVIRONMENT.SIMULATION THEN
				GVL_TWO_PALLET.astSimulationConfig[uiTwin] := stTwinRequest.Config;
			ELSE
				GVL_TWO_PALLET.astConfig[uiTwin] := stTwinRequest.Config;
			END_IF;
			axTwinConfigurationChanged[uiTwin] := TRUE;
			uiTwinRequestResult := UINT#1;
		END_IF;
	ELSIF ((uiTwinPallet = 1) AND GVL_TWO_PALLET.astStatus[uiTwin].xEdit1Allowed)
		OR ((uiTwinPallet = 2) AND GVL_TWO_PALLET.astStatus[uiTwin].xEdit2Allowed) THEN
		CASE stTwinRequest.uiCommand OF
			20: GVL_TWO_PALLET.astStore[uiTwin].axLoaded[uiTwinPallet] := TRUE; uiTwinRequestResult := 1;
			21, 22:
				FOR uiTwinSlot := 1 TO 96 DO
					GVL_TWO_PALLET.astStore[uiTwin].astPallet[uiTwinPallet].aSlots[uiTwinSlot].xInPosition := stTwinRequest.uiCommand = 22;
					GVL_TWO_PALLET.astStore[uiTwin].astPallet[uiTwinPallet].aSlots[uiTwinSlot].eDetailType := E_DETAIL_TYPE.NONE;
					GVL_TWO_PALLET.astStore[uiTwin].astPallet[uiTwinPallet].aSlots[uiTwinSlot].uiProductType := 0;
					IF stTwinRequest.uiCommand = 22 THEN
						GVL_TWO_PALLET.astStore[uiTwin].astPallet[uiTwinPallet].aSlots[uiTwinSlot].eDetailType := E_DETAIL_TYPE.BLANK;
						GVL_TWO_PALLET.astStore[uiTwin].astPallet[uiTwinPallet].aSlots[uiTwinSlot].uiProductType := GVL_MULTI_TYPE.Config.auiSlotType[uiTwinSlot];
					END_IF;
				END_FOR;
				GVL_TWO_PALLET.astStore[uiTwin].axLoaded[uiTwinPallet] := FALSE; uiTwinRequestResult := 1;
			23:
				IF (stTwinRequest.uiSlot >= 1) AND (stTwinRequest.uiSlot <= 96) AND (stTwinRequest.uiContent <= 2)
					AND ((stTwinRequest.uiContent = 0) OR ((stTwinRequest.uiProductType >= 1) AND (stTwinRequest.uiProductType <= GVL_MULTI_TYPE.Config.uiTypeCount))) THEN
					uiTwinSlot := stTwinRequest.uiSlot;
					GVL_TWO_PALLET.astStore[uiTwin].astPallet[uiTwinPallet].aSlots[uiTwinSlot].xInPosition := stTwinRequest.uiContent <> 0;
					CASE stTwinRequest.uiContent OF
						0: GVL_TWO_PALLET.astStore[uiTwin].astPallet[uiTwinPallet].aSlots[uiTwinSlot].eDetailType := E_DETAIL_TYPE.NONE;
						1: GVL_TWO_PALLET.astStore[uiTwin].astPallet[uiTwinPallet].aSlots[uiTwinSlot].eDetailType := E_DETAIL_TYPE.BLANK;
						2: GVL_TWO_PALLET.astStore[uiTwin].astPallet[uiTwinPallet].aSlots[uiTwinSlot].eDetailType := E_DETAIL_TYPE.DETAIL;
					END_CASE;
					GVL_TWO_PALLET.astStore[uiTwin].astPallet[uiTwinPallet].aSlots[uiTwinSlot].uiProductType := stTwinRequest.uiProductType;
					GVL_TWO_PALLET.astStore[uiTwin].axLoaded[uiTwinPallet] := FALSE; uiTwinRequestResult := 1;
				END_IF;
		END_CASE;
	END_IF;
END_IF;
IF uiTwinRequestResult <> 0 THEN
	GVL_HMI.uiTwinResult := uiTwinRequestResult;
	GVL_HMI.udiTwinAckSeq := udiTwinSnapshot;
	IF uiTwinRequestResult <> 1 THEN
		uiTwin := LIMIT(UINT#1, stTwinRequest.uiMagazine, UINT#2);
		// Команды механизма 1..19 и 25..28 уже формируют предупреждение внутри FB в этом же скане.
		IF GVL_TWO_PALLET.auiCommand[uiTwin] <> stTwinRequest.uiCommand THEN
			axTwinExternalCommandRejected[uiTwin] := TRUE;
		END_IF;
	END_IF;
END_IF;

GVL_CELL_SETTINGS.MagazineRows := 12;
GVL_CELL_SETTINGS.MagazineColumns := 10;
IF GVL_TWO_PALLET.uiMode = 1 THEN GVL_CELL_SETTINGS.MagazineRows := 12; GVL_CELL_SETTINGS.MagazineColumns := 8; END_IF;
GVL_HMI.MagazineRows := GVL_CELL_SETTINGS.MagazineRows;
GVL_HMI.MagazineColumns := GVL_CELL_SETTINGS.MagazineColumns;
FOR uiTwin := 1 TO 2 DO
	IF GVL_TWO_PALLET.uiMode = 1 THEN
		uiTwinPallet := GVL_TWO_PALLET.astStatus[uiTwin].uiRobotPallet;
		IF (uiTwinPallet < UINT#1) OR (uiTwinPallet > UINT#2) THEN
			uiTwinPallet := UINT#1;
		END_IF;
		GVL_DETAIL.astMagazine[uiTwin] := GVL_TWO_PALLET.astStore[uiTwin].astPallet[uiTwinPallet];
	END_IF;
END_FOR;

(* ---- PLC_PRG.RunTwoPalletAxis.st ---- *)
METHOD PRIVATE RunTwoPalletAxis

// --- BEGIN IMPLEMENTATION ---

// Используем две существующие виртуальные SoftMotion-оси прежних магазинов.
// Ссылки назначаются каждый скан до проверки __ISVALIDREF и вызова FB_AXIS.
GVL_TWO_PALLET.Axis1 REF= Magazine_1;
GVL_TWO_PALLET.Axis2 REF= Magazine_2;
GVL_TWO_PALLET.astInput[1].xAxisBound := __ISVALIDREF(GVL_TWO_PALLET.Axis1);
GVL_TWO_PALLET.astInput[2].xAxisBound := __ISVALIDREF(GVL_TWO_PALLET.Axis2);
FOR uiTwin := 1 TO 2 DO
	GVL_TWO_PALLET.astAxis[uiTwin].Command.xEnable := GVL_TWO_PALLET.astOutput[uiTwin].xPowerOn;
	GVL_TWO_PALLET.astAxis[uiTwin].Command.xDisable := GVL_TWO_PALLET.astOutput[uiTwin].xPowerOff
		OR (GVL_TWO_PALLET.uiMode = 0);
	GVL_TWO_PALLET.astAxis[uiTwin].Command.xPowerPermit := (GVL_TWO_PALLET.uiMode = 1)
		AND CELL_SAFETY.Status.xReady AND GVL_TWO_PALLET.astInput[uiTwin].xIoMapped;
	GVL_TWO_PALLET.astAxis[uiTwin].Command.xGlobalError := GVL_CELL_CONTROL.xGlobalError;
	GVL_TWO_PALLET.astAxis[uiTwin].Command.xResetAllError := GVL_TWO_PALLET.astOutput[uiTwin].xDriveReset;
	GVL_TWO_PALLET.astAxis[uiTwin].Command.xStop := GVL_TWO_PALLET.astOutput[uiTwin].xStop;
	GVL_TWO_PALLET.astAxis[uiTwin].Command.xHome := GVL_TWO_PALLET.astOutput[uiTwin].xHome;
	GVL_TWO_PALLET.astAxis[uiTwin].Command.xMoveAbsolute := GVL_TWO_PALLET.astOutput[uiTwin].xMove;
	GVL_TWO_PALLET.astAxis[uiTwin].Command.xJogPositive := GVL_TWO_PALLET.astOutput[uiTwin].xJogPositive;
	GVL_TWO_PALLET.astAxis[uiTwin].Command.xJogNegative := GVL_TWO_PALLET.astOutput[uiTwin].xJogNegative;
	GVL_TWO_PALLET.astAxis[uiTwin].MotionParam.lrTargetPosition := GVL_TWO_PALLET.astOutput[uiTwin].lrTarget;
	GVL_TWO_PALLET.astAxis[uiTwin].MotionParam.lrHomePosition := GVL_TWO_PALLET.astActiveConfig[uiTwin].lrHome;
	GVL_TWO_PALLET.astAxis[uiTwin].MotionParam.lrVelocity := GVL_TWO_PALLET.astActiveConfig[uiTwin].lrVelocity;
	GVL_TWO_PALLET.astAxis[uiTwin].MotionParam.lrAcceleration := GVL_TWO_PALLET.astActiveConfig[uiTwin].lrAcceleration;
	GVL_TWO_PALLET.astAxis[uiTwin].MotionParam.lrDeceleration := GVL_TWO_PALLET.astActiveConfig[uiTwin].lrDeceleration;
	GVL_TWO_PALLET.astAxis[uiTwin].MotionParam.lrJerk := GVL_TWO_PALLET.astActiveConfig[uiTwin].lrJerk;
	GVL_TWO_PALLET.astAxis[uiTwin].Timeouts := GVL_CELL_SETTINGS.stAxisTimeouts;
	GVL_TWO_PALLET.astAxis[uiTwin].Timeouts.tHomeTimeout := GVL_TWO_PALLET.astActiveConfig[uiTwin].tHome;
	GVL_TWO_PALLET.astAxis[uiTwin].Timeouts.tMoveTimeout := GVL_TWO_PALLET.astActiveConfig[uiTwin].tMove;
END_FOR;
IF __ISVALIDREF(GVL_TWO_PALLET.Axis1) THEN
	TWIN_AXIS_1(Axis := GVL_TWO_PALLET.Axis1, AxisData := GVL_TWO_PALLET.astAxis[1],
		xResetPermit := GVL_CELL_CONTROL.xManual AND NOT GVL_CELL_MANAGER.Status.xRunning);
END_IF;
IF __ISVALIDREF(GVL_TWO_PALLET.Axis2) THEN
	TWIN_AXIS_2(Axis := GVL_TWO_PALLET.Axis2, AxisData := GVL_TWO_PALLET.astAxis[2],
		xResetPermit := GVL_CELL_CONTROL.xManual AND NOT GVL_CELL_MANAGER.Status.xRunning);
END_IF;
FOR uiTwin := 1 TO 2 DO
	GVL_TWO_PALLET.astInput[uiTwin].xPowered := GVL_TWO_PALLET.astAxis[uiTwin].Status.xPowered;
	GVL_TWO_PALLET.astInput[uiTwin].xHomed := GVL_TWO_PALLET.astAxis[uiTwin].Status.xHomed;
	GVL_TWO_PALLET.astInput[uiTwin].xStandstill := GVL_TWO_PALLET.astAxis[uiTwin].Status.xStandstill;
	GVL_TWO_PALLET.astInput[uiTwin].xDriveError := GVL_TWO_PALLET.astAxis[uiTwin].Status.xError;
	GVL_TWO_PALLET.astInput[uiTwin].xMotionDone := GVL_TWO_PALLET.astAxis[uiTwin].Status.xDone;
	GVL_TWO_PALLET.astInput[uiTwin].lrPosition := GVL_TWO_PALLET.astAxis[uiTwin].Status.lrActualPosition;
	TWIN_SIM[uiTwin](
		xEnable := (GVL_TWO_PALLET.uiMode = UINT#1)
			AND (GVL_CELL_SETTINGS.eTestEnvironment = E_CELL_TEST_ENVIRONMENT.SIMULATION),
		uiP1Signals := GVL_TWO_PALLET.astActiveConfig[uiTwin].uiP1Signals,
		Command := GVL_TWO_PALLET.astOutput[uiTwin]);
	IF (GVL_TWO_PALLET.uiMode = UINT#1)
		AND (GVL_CELL_SETTINGS.eTestEnvironment = E_CELL_TEST_ENVIRONMENT.SIMULATION) THEN
		GVL_TWO_PALLET.astInput[uiTwin].xIoMapped := TRUE;
		GVL_TWO_PALLET.astInput[uiTwin].xLiftDown := TWIN_SIM[uiTwin].xLiftDown;
		GVL_TWO_PALLET.astInput[uiTwin].xLiftUp := TWIN_SIM[uiTwin].xLiftUp;
		GVL_TWO_PALLET.astInput[uiTwin].xLockIn := TWIN_SIM[uiTwin].xLockIn;
		GVL_TWO_PALLET.astInput[uiTwin].xLockOut := TWIN_SIM[uiTwin].xLockOut;
		GVL_TWO_PALLET.astInput[uiTwin].xStopIn := TWIN_SIM[uiTwin].xStopIn;
		GVL_TWO_PALLET.astInput[uiTwin].xStopOut := TWIN_SIM[uiTwin].xStopOut;
		GVL_TWO_PALLET.astInput[uiTwin].xLimitNegative := FALSE;
		GVL_TWO_PALLET.astInput[uiTwin].xLimitPositive := FALSE;
		GVL_TWO_PALLET.astInput[uiTwin].xHomeSensor := GVL_TWO_PALLET.astInput[uiTwin].xHomed
			AND (ABS(GVL_TWO_PALLET.astInput[uiTwin].lrPosition
				- GVL_TWO_PALLET.astActiveConfig[uiTwin].lrHome)
				<= GVL_TWO_PALLET.astActiveConfig[uiTwin].lrTolerance);
		axTwinSimIoOwned[uiTwin] := TRUE;
	ELSIF axTwinSimIoOwned[uiTwin] THEN
		// После выхода из виртуальной среды не оставляем её герконы как реальные.
		GVL_TWO_PALLET.astInput[uiTwin].xIoMapped := FALSE;
		GVL_TWO_PALLET.astInput[uiTwin].xLiftDown := FALSE;
		GVL_TWO_PALLET.astInput[uiTwin].xLiftUp := FALSE;
		GVL_TWO_PALLET.astInput[uiTwin].xLockIn := FALSE;
		GVL_TWO_PALLET.astInput[uiTwin].xLockOut := FALSE;
		GVL_TWO_PALLET.astInput[uiTwin].xStopIn := FALSE;
		GVL_TWO_PALLET.astInput[uiTwin].xStopOut := FALSE;
		GVL_TWO_PALLET.astInput[uiTwin].xLimitNegative := FALSE;
		GVL_TWO_PALLET.astInput[uiTwin].xLimitPositive := FALSE;
		GVL_TWO_PALLET.astInput[uiTwin].xHomeSensor := FALSE;
		axTwinSimIoOwned[uiTwin] := FALSE;
	END_IF;
END_FOR;

(* ---- PLC_PRG.SetApplicationDefaults.st ---- *)
METHOD PRIVATE SetApplicationDefaults

// --- BEGIN IMPLEMENTATION ---

// При старте PLC ячейка всегда включается в ручном режиме: автоматический цикл
// требует явного переключения оператором. Однократный флаг также повторно
// применяет безопасные значения при Online Change, когда initializer GVL
// может не перезаписать уже существующее значение. Инициализация выполняется до
// RunCellControl, чтобы автомат не увидел прежние настройки даже на один цикл.
IF NOT xApplicationStartupInitialized THEN
	GVL_CELL_CONTROL.xManual := TRUE;
	FOR uiMachine := 1 TO 3 DO
		GVL_HMI.axMachineUsed[uiMachine] := FALSE;
	END_FOR;
	// RETAIN uiMode переживает перезапуск PLC, поэтому явно выбираем двухпалетный
	// тип на старте. При реальной смене типа старые базы магазинов недействительны.
	IF GVL_TWO_PALLET.uiMode <> UINT#1 THEN
		GVL_TWO_PALLET.uiMode := UINT#1;
		GVL_POINT.astRetainPoints[UINT#14].xConfigured := FALSE;
		GVL_POINT.astRetainPoints[UINT#15].xConfigured := FALSE;
		xPointTableReady := FALSE;
	END_IF;
	GVL_CELL_SETTINGS.eTestEnvironment := E_CELL_TEST_ENVIRONMENT.SIMULATION;
	xApplicationStartupInitialized := TRUE;
END_IF;

// При первом запуске этой схемы намеренно отбрасываем прежние инженерные
// координаты. Нулевая скорость и xConfigured=FALSE не позволяют принять
// нулевую точку за пригодную для движения.
IF GVL_POINT.udiPointStorageVersion <> GVL_POINT.udiExpectedPointStorageVersion THEN
	FOR uiPointEditorIndex := UINT#1 TO INT_TO_UINT(GVL_POINT.iPersistentPointCapacity) DO
		GVL_POINT.astRetainPoints[uiPointEditorIndex].Name := '';
		GVL_POINT.astRetainPoints[uiPointEditorIndex].X := 0.0;
		GVL_POINT.astRetainPoints[uiPointEditorIndex].Y := 0.0;
		GVL_POINT.astRetainPoints[uiPointEditorIndex].Z := 0.0;
		GVL_POINT.astRetainPoints[uiPointEditorIndex].MagazineSafeZ := 0.0;
		GVL_POINT.astRetainPoints[uiPointEditorIndex].MagazineChangeZ := 0.0;
		GVL_POINT.astRetainPoints[uiPointEditorIndex].SpeedFactor := 0.0;
		GVL_POINT.astRetainPoints[uiPointEditorIndex].xConfigured := FALSE;
	END_FOR;
	GVL_POINT.udiPointStorageVersion := GVL_POINT.udiExpectedPointStorageVersion;
END_IF;

// Единственное соответствие компактного редакторского индекса, стабильного
// E_POINT_NAME и прежнего индекса Persistent-массива. Три legacy-точки INSIDE
// пропущены; рецепты станков их не используют.
xPointTableReady := TRUE;
FOR uiPointEditorIndex := UINT#1 TO INT_TO_UINT(GVL_POINT.iEditablePointCount) DO
	uiPointStorageIndex := UINT#0;
	CASE uiPointEditorIndex OF
		UINT#1: ePointEditorName := E_POINT_NAME.MACHINE_1_ABOVE; uiPointStorageIndex := UINT#1;
		UINT#2: ePointEditorName := E_POINT_NAME.MACHINE_1_CHUCK_APROACH; uiPointStorageIndex := UINT#3;
		UINT#3: ePointEditorName := E_POINT_NAME.MACHINE_1_CHUCK_POSITION; uiPointStorageIndex := UINT#4;
		UINT#4: ePointEditorName := E_POINT_NAME.MACHINE_2_ABOVE; uiPointStorageIndex := UINT#5;
		UINT#5: ePointEditorName := E_POINT_NAME.MACHINE_2_CHUCK_APROACH; uiPointStorageIndex := UINT#7;
		UINT#6: ePointEditorName := E_POINT_NAME.MACHINE_2_CHUCK_POSITION; uiPointStorageIndex := UINT#8;
		UINT#7: ePointEditorName := E_POINT_NAME.MACHINE_3_ABOVE; uiPointStorageIndex := UINT#9;
		UINT#8: ePointEditorName := E_POINT_NAME.MACHINE_3_CHUCK_APROACH; uiPointStorageIndex := UINT#11;
		UINT#9: ePointEditorName := E_POINT_NAME.MACHINE_3_CHUCK_POSITION; uiPointStorageIndex := UINT#12;
		UINT#10: ePointEditorName := E_POINT_NAME.HOME_SAFETY; uiPointStorageIndex := UINT#13;
		UINT#11: ePointEditorName := E_POINT_NAME.MAGAZINE_1_DETAIL; uiPointStorageIndex := UINT#14;
		UINT#12: ePointEditorName := E_POINT_NAME.MAGAZINE_2_DETAIL; uiPointStorageIndex := UINT#15;
	ELSE
		ePointEditorName := E_POINT_NAME.NONE;
	END_CASE;

	IF (ePointEditorName <> E_POINT_NAME.NONE) AND (uiPointStorageIndex <> UINT#0) THEN
		GVL_POINT.Points[ePointEditorName] := GVL_POINT.astRetainPoints[uiPointStorageIndex];
		IF (ePointEditorName = E_POINT_NAME.MAGAZINE_1_DETAIL)
		OR (ePointEditorName = E_POINT_NAME.MAGAZINE_2_DETAIL) THEN
			GVL_POINT.Points[ePointEditorName].xConfigured :=
				GVL_POINT.astRetainPoints[uiPointStorageIndex].xConfigured
				AND (GVL_POINT.astRetainPoints[uiPointStorageIndex].MagazineSafeZ <> LREAL#0.0)
				AND (GVL_POINT.astRetainPoints[uiPointStorageIndex].MagazineChangeZ <> LREAL#0.0);
		END_IF;
		IF NOT GVL_POINT.Points[ePointEditorName].xConfigured THEN
			xPointTableReady := FALSE;
		END_IF;
	ELSE
		xPointTableReady := FALSE;
	END_IF;
END_FOR;

(* ---- PLC_PRG.st ---- *)
PROGRAM PLC_PRG
VAR
	AXIS_X         : FB_AXIS; // Управление осью X
	AXIS_Y         : FB_AXIS; // Управление осью Y
	AXIS_Z         : FB_AXIS; // Управление осью Z
	GROUP_XYZ      : FB_AXIS_GROUP; // Управление группой осей XYZ
	HMI            : FB_HMI; // Обмен данными с визуализацией
	MOTION_MANAGER : FB_MOTION_MANAGER; // Менеджер движения по именованным точкам
	MACHINE_1      : FB_MACHINE; // Логика первого станка
	MACHINE_2      : FB_MACHINE; // Логика второго станка
	MACHINE_3      : FB_MACHINE; // Логика третьего станка
	MACHINE_1_SIM  : FB_MACHINE_SIMULATION; // Симуляция первого станка
	MACHINE_2_SIM  : FB_MACHINE_SIMULATION; // Симуляция второго станка
	MACHINE_3_SIM  : FB_MACHINE_SIMULATION; // Симуляция третьего станка
	MAGAZINE       : FB_MAGAZINE; // Управление магазином деталей
	ROBOT          : FB_ROBOT; // Координация движений и захвата робота
END_VAR

// --- BEGIN IMPLEMENTATION ---

//Над станком 1
GVL_POINT.Points[E_POINT_NAME.MACHINE_1_ABOVE].X := 425;
GVL_POINT.Points[E_POINT_NAME.MACHINE_1_ABOVE].Y := 100;
GVL_POINT.Points[E_POINT_NAME.MACHINE_1_ABOVE].Z := 216;
GVL_POINT.Points[E_POINT_NAME.MACHINE_1_ABOVE].SpeedFactor := 1.0;

//В станке 1
GVL_POINT.Points[E_POINT_NAME.MACHINE_1_INSIDE].X := 425;
GVL_POINT.Points[E_POINT_NAME.MACHINE_1_INSIDE].Y := 100;
GVL_POINT.Points[E_POINT_NAME.MACHINE_1_INSIDE].Z := 458;
GVL_POINT.Points[E_POINT_NAME.MACHINE_1_INSIDE].SpeedFactor := 1.0;

//У патрона 1
GVL_POINT.Points[E_POINT_NAME.MACHINE_1_CHUCK_APROACH].X := 425;
GVL_POINT.Points[E_POINT_NAME.MACHINE_1_CHUCK_APROACH].Y := 100;
GVL_POINT.Points[E_POINT_NAME.MACHINE_1_CHUCK_APROACH].Z := 506;
GVL_POINT.Points[E_POINT_NAME.MACHINE_1_CHUCK_APROACH].SpeedFactor := 1.0;

//В патроне 1
GVL_POINT.Points[E_POINT_NAME.MACHINE_1_CHUCK_POSITION].X := 378;
GVL_POINT.Points[E_POINT_NAME.MACHINE_1_CHUCK_POSITION].Y := 100;
GVL_POINT.Points[E_POINT_NAME.MACHINE_1_CHUCK_POSITION].Z := 506;
GVL_POINT.Points[E_POINT_NAME.MACHINE_1_CHUCK_POSITION].SpeedFactor := 1.0;

GVL_AXIS.arrAxis[1].Command.xGlobalError := GVL_CELL_CONTROL.xGlobalError;
GVL_AXIS.arrAxis[2].Command.xGlobalError := GVL_CELL_CONTROL.xGlobalError;
GVL_AXIS.arrAxis[3].Command.xGlobalError := GVL_CELL_CONTROL.xGlobalError;

GVL_AXIS.arrAxis[1].Command.xResetAllError := GVL_CELL_CONTROL.xReset;
GVL_AXIS.arrAxis[2].Command.xResetAllError := GVL_CELL_CONTROL.xReset;
GVL_AXIS.arrAxis[3].Command.xResetAllError := GVL_CELL_CONTROL.xReset;

GVL_AXIS_GROUP.AxisGroup.Command.xGlobalError := GVL_CELL_CONTROL.xGlobalError;
GVL_AXIS_GROUP.AxisGroup.Command.xReset := GVL_CELL_CONTROL.xReset;

AXIS_X(
	Axis:= X,
	AxisData := GVL_AXIS.arrAxis[1]
);

AXIS_Y(
	Axis:= Y,
	AxisData := GVL_AXIS.arrAxis[2]
);

AXIS_Z(
	Axis:= Z,
	AxisData := GVL_AXIS.arrAxis[3]
);

GROUP_XYZ(
	AxisGroup :=AXIS_GROUP,
	GroupData :=GVL_AXIS_GROUP.AxisGroup
);

HMI(
	GroupData := GVL_AXIS_GROUP.AxisGroup,
	HMI := GVL_HMI.HMI
);

MACHINE_1.stPoints.eAbove := E_POINT_NAME.MACHINE_1_ABOVE;
MACHINE_1.stPoints.eChuck := E_POINT_NAME.MACHINE_1_CHUCK_POSITION;
MACHINE_1.stPoints.eChuckApproach := E_POINT_NAME.MACHINE_1_CHUCK_APROACH;
MACHINE_1.stPoints.eInside := E_POINT_NAME.MACHINE_1_INSIDE;
MACHINE_1.stPoints.eNone := E_POINT_NAME.NONE;

MACHINE_1(
	xResetGlobal := GVL_CELL_CONTROL.xReset,
	xGlobalError := GVL_CELL_CONTROL.xGlobalError,
	stChangeRecipe := GVL_CELL_SETTINGS.CHANGE_MACHINE,
	stMachineStatus := MACHINE_1_SIM.Status,
	stRobotStatus := ROBOT.Status
);

MACHINE_2.stPoints.eAbove := E_POINT_NAME.MACHINE_2_ABOVE;
MACHINE_2.stPoints.eChuck := E_POINT_NAME.MACHINE_2_CHUCK_POSITION;
MACHINE_2.stPoints.eChuckApproach := E_POINT_NAME.MACHINE_2_CHUCK_APROACH;
MACHINE_2.stPoints.eInside := E_POINT_NAME.MACHINE_2_INSIDE;
MACHINE_2.stPoints.eNone := E_POINT_NAME.NONE;

MACHINE_2(
	xResetGlobal := GVL_CELL_CONTROL.xReset,
	xGlobalError := GVL_CELL_CONTROL.xGlobalError,
	stChangeRecipe := GVL_CELL_SETTINGS.CHANGE_MACHINE,
	stMachineStatus := MACHINE_2_SIM.Status,
	stRobotStatus := ROBOT.Status
);

MACHINE_3.stPoints.eAbove := E_POINT_NAME.MACHINE_3_ABOVE;
MACHINE_3.stPoints.eChuck := E_POINT_NAME.MACHINE_3_CHUCK_POSITION;
MACHINE_3.stPoints.eChuckApproach := E_POINT_NAME.MACHINE_3_CHUCK_APROACH;
MACHINE_3.stPoints.eInside := E_POINT_NAME.MACHINE_3_INSIDE;
MACHINE_3.stPoints.eNone := E_POINT_NAME.NONE;

MACHINE_3(
	xResetGlobal := GVL_CELL_CONTROL.xReset,
	xGlobalError := GVL_CELL_CONTROL.xGlobalError,
	stChangeRecipe := GVL_CELL_SETTINGS.CHANGE_MACHINE,
	stMachineStatus := MACHINE_3_SIM.Status,
	stRobotStatus := ROBOT.Status
);

MACHINE_1_SIM(
	Command := MACHINE_1.Command.stIo
);

MACHINE_2_SIM(
	Command := MACHINE_2.Command.stIo
);

MACHINE_3_SIM(
	Command := MACHINE_3.Command.stIo
);

MAGAZINE(
	stRobotStatus := ROBOT.Status,
	stMagazineCommand := GVL_ROBOT.stMagazineAutoCommand,
	stHmiCommand := GVL_HMI.HMI.Command.stRobot,
	xManual := GVL_CELL_CONTROL.xManual,
	xReset := GVL_CELL_CONTROL.xReset,
	xGlobalError := GVL_CELL_CONTROL.xGlobalError,
	xMode := GVL_HMI.HMI.Command.xModbusMode,
	xHmiEnable := GVL_HMI.HMI.Command.xMagazineEnable,
	xHmiDisable := GVL_HMI.HMI.Command.xMagazineDisable,
	uiRows := GVL_CELL_SETTINGS.MagazineRows,
	uiColumns := GVL_CELL_SETTINGS.MagazineColumns,
	lrPitchX := GVL_CELL_SETTINGS.MagazinePitchX,
	lrPitchY := GVL_CELL_SETTINGS.MagazinePitchY,
	lrSafeZ := GVL_CELL_SETTINGS.MagazineSafeZ,
	stDetail := GVL_DETAIL.arrDetail,
	stPoint := GVL_POINT.Points
);

ROBOT(
	stMachine_1_command := MACHINE_1.Command.stRobot,
	stMachine_2_command := MACHINE_2.Command.stRobot,
	stMachine_3_command := MACHINE_3.Command.stRobot,
	stMagazineCommand := MAGAZINE.Command,
	stHmiCommand := GVL_HMI.HMI.Command.stRobot,
	xReset := GVL_CELL_CONTROL.xReset,
	xManual := GVL_CELL_CONTROL.xManual,
	xMode := GVL_HMI.HMI.Command.xModbusMode,
	xGlobalError := GVL_CELL_CONTROL.xGlobalError,
	xModbusBusy := GVL_ROBOT.xModbusBusy,
	xModbusDone := GVL_ROBOT.xModbusDone,
	xModbusError := GVL_ROBOT.xModbusError,

    stPoint := GVL_POINT.Points,

    stMotionManager := GVL_MOTION_MANAGER.stMotionManager,
    GroupData := GVL_AXIS_GROUP.AxisGroup,
    stPointManager := GVL_POINT_MANAGER.PointManager
);

GVL_ROBOT.stModbusCommand := ROBOT.ModbusCommand;

(* ---- STATISTIC.st ---- *)
PROGRAM STATISTIC
VAR
	fb_Statistic : FB_STATISTIC;
END_VAR

// --- BEGIN IMPLEMENTATION ---

fb_Statistic(
	xStart          := GVL_CELL_MANAGER.Status.xRunning,
	uiSimulationTimeFactor := GVL_CELL_SETTINGS.uiSimulationTimeFactorApplied,
	eActiveAction 	:= GVL_ROBOT.Diag.eActiveAction,
	eActivePoint  	:= GVL_ROBOT.Diag.eActivePoint,
	xBusyMagazine 	:= GVL_MAGAZINE.astStatus[1].xBusy OR GVL_MAGAZINE.astStatus[2].xBusy,
	xBusyMachine_1 	:= GVL_MACHINE.Status[1].xBusy,
	xBusyMachine_2 	:= GVL_MACHINE.Status[2].xBusy,
	xBusyMachine_3 	:= GVL_MACHINE.Status[3].xBusy,
	xCycleActiveMachine_1 	:= GVL_MACHINE.Status[1].stIo.xCycleActive,
	xCycleActiveMachine_2 	:= GVL_MACHINE.Status[2].stIo.xCycleActive,
	xCycleActiveMachine_3 	:= GVL_MACHINE.Status[3].stIo.xCycleActive,
	xBusyRobot 		:=	GVL_ROBOT.Status.xBusy,
	stStatistic     =>  GVL_STATISTIC.stStatistic
);
